// Jidien Kachu Edited in 2025/10/14
FUNCTION_BLOCK FB_RobotAbsMove_V2 EXTENDS FB_ObjectBase_V2 IMPLEMENTS IBasicElement
VAR_INPUT
    Robot         				: REFERENCE TO FB_FanucRobot_Basic_V2;
    LowerConveyor 				: REFERENCE TO FB_Motor;
    // Command   : ST_WareHouseWithRobotMove_Command;
    Info 						: st_AutoSixAxisAbsMoveParameter;
	Input 						: ST_InputTable;
    Stop 						: BOOL;
	Output 						: ST_OutputTable;
	Cylinder 					: REFERENCE TO UNI_CylinderList;
	bCheckUpperCV_ServiceDone	: BOOL;
END_VAR
VAR_OUTPUT
    // Status : ST_WareHouseWithRobotMove_Status;
	AClampMoveDone	: BOOL;
	BClampMoveDone	: BOOL;
END_VAR
VAR
    //_Abort       : BOOL;
    strStatus    : STRING;
    uiResumeStep : UINT;

    Area : E_RobotArea;
    UseA : BOOL;
    UseB : BOOL;

    Get                         : BOOL;
    tonTimeOut                  : TON;
	bTimeOutIN					: BOOL;
	tonDelay					 : TON;
    _UniqueErrorCode            : STRING;
    FirstSensorOfLowerConveyor  : BOOL;
    SecondSensorOfLowerConveyor : BOOL;

	//Added by Jidien Kachu in 2025/10/09
	uiLastBothStep	: UINT;
	uiLastSingleClampStep	: UINT;
	bRobotTimeOutIN	: BOOL;
	tonRobotTimeOut	: TON;
	uiBothStep	: UINT;
	uiSingleClampStep	: UINT;
	bMotorDelayIN	: BOOL;
	tonMotorDelay	: TON;
	bIOTimeoutIN	: BOOL;
	tonIOTimeout	: TON;
	bRetry: BOOL;
	
	//Added by Gamin in 2025//11/24
	_AClampDoingWork	: BOOL;
	_BClampDoingWork	: BOOL;
END_VAR

SUPER^.A10_StateControl();
A00_BasicUnits();
FirstSensorOfLowerConveyor := Input.bLowCV_BoxArrived_Sensor;
SecondSensorOfLowerConveyor := NOT Input.bLowCV_2ndBoxGap_Sensor;// .bLowCV_Block2Detect_Sensor;

(*============================================================
Create Date : 2025/11/22
Last Update	: 2026/04/01
Change Log  : 2025/11/24，send flag A clamp done and B clamp done for C# use to SQL // Edited : Gamin
			  2026/04/01，移植泰興鏡射機版本。
============================================================*)

ACTION A00_BasicUnits:
tonTimeOut(IN:= bTimeOutIN AND NOT THIS^.Stop, PT:=T#60S);
tonDelay(PT:=T#1S);
ErrorID :=2200;
tonMotorDelay(IN:= bMotorDelayIN,PT:=T#1S);
tonIOTimeout(IN:= bIOTimeoutIN,PT:= T#1S);
END_ACTION

METHOD M_CheckClampStatus : BOOL
VAR_INPUT
END_VAR
M_CheckClampStatus := FALSE;

IF NOT UseA AND NOT UseB THEN
	M_CheckClampStatus 	:= FALSE;
	strStatus 			:= 'FB_RobotAbsMove_V2 ,Wrong Command , Both Clammp not used';
	RETURN;
END_IF

IF UseA THEN
	IF Get THEN
		IF NOT Robot._DI1.ClampA_Open THEN
			M_CheckClampStatus  := FALSE;
			strStatus			:= 'FB_RobotAbsMove_V2 ,Robot Use A Clamp Get ,but Clamp not open ';
			RETURN;
		END_IF
	ELSE
		IF Robot._DI1.ClampA_Open THEN
			M_CheckClampStatus	:= FALSE;
			strStatus			:= 'FB_RobotAbsMove_V2 ,Robot Use A Clamp Place ,but Clamp open';
			RETURN;
		END_IF
	END_IF
END_IF
IF UseB THEN
	IF Get THEN
		IF NOT Robot._DI1.ClampB_Open THEN
			M_CheckClampStatus  := FALSE;
			strStatus			:= 'FB_RobotAbsMove_V2 ,Robot Use B Clamp Get ,but Clamp not open ';
			RETURN;
		END_IF
	ELSE
		IF Robot._DI1.ClampB_Open THEN
			M_CheckClampStatus	:= FALSE;
			strStatus			:= 'FB_RobotAbsMove_V2 ,Robot Use B Clamp Place ,but Clamp open';
			RETURN;
		END_IF
	END_IF
END_IF

M_CheckClampStatus := TRUE;
END_METHOD

METHOD M_CheckCommand : BOOL // True : Command is useful
VAR_INPUT
END_VAR
VAR
	
END_VAR
// Check command paremeter is correct


IF Info.A_Get <> Info.B_Get THEN
	strStatus:='Wrong command ,GetA not match to GetB';
	M_CheckCommand:=FALSE;
	RETURN;
ELSE		
	THIS^.Get :=Info.A_Get;
END_IF

IF Info.A_Area<> Info.B_Area THEN
	IF NOT(Info.A_Area=99 OR Info.B_Area=99) THEN
	strStatus:='Wrong command ,Area A not match to Area B';
	M_CheckCommand:=FALSE;
	RETURN;
END_IF
END_IF

IF Info.A_Area = 99 AND Info.B_Area = 99 THEN
	strStatus:='Wrong command ,Both Area are 99';
	M_CheckCommand:=FALSE;
	RETURN;
END_IF

CASE LREAL_TO_INT(Info.A_Area) OF
	1 : //Normal command : RoundBelt
		IF Info.A_Position<1 OR  Info.A_Position>3 THEN
			strStatus:='Wrong command ,Position A Not allow';
			M_CheckCommand:=FALSE;
			RETURN;	
		ELSE
			Area := E_RobotArea.RoundBelt;
			UseA :=TRUE	;	
		END_IF
		
	2:	//Buffer area
		IF Info.A_Position<1 OR  Info.A_Position>40 THEN
			strStatus:='Wrong command ,Position A Not allow';
			M_CheckCommand:=FALSE;
			RETURN;	
		ELSE
			Area := E_RobotArea.BufferArea;
			UseA :=TRUE	;	
		END_IF
	3: //Allocated/Empty conveyor
		IF Info.A_Position<1 OR  Info.A_Position>2 THEN
			strStatus:='Wrong command ,Position A Not allow';
			M_CheckCommand:=FALSE;
			RETURN;	
		ELSE
			Area := E_RobotArea.TransmitCV;
			UseA :=TRUE	;	
		END_IF
	5: //FeedIn/Out conveyor
		IF Info.A_Position<1 OR  Info.A_Position>5 THEN
			strStatus:='Wrong command ,Position A Not allow';
			M_CheckCommand:=FALSE;
			RETURN;	
		ELSIF Info.A_Position=3 AND Get THEN
			strStatus:='Wrong command ,Can Not Get box from FeedOut conveyor ';
			M_CheckCommand:=FALSE;
			RETURN;	
		ELSE
			Area := E_RobotArea.InOutConveyor;
			UseA :=TRUE	;	
		END_IF
	7: // PullOut conveyor
		IF Info.A_Position<1 OR  Info.A_Position>2 THEN
			strStatus:='Wrong command ,Position A Not allow';
			M_CheckCommand:=FALSE;
			RETURN;	
		ELSE
			Area := E_RobotArea.PullOutConveyor;
			UseA :=TRUE	;	
		END_IF
	
	99: //ClampA not use
		UseA :=FALSE;
	
	ELSE //Wrong command
		strStatus:='Wrong command ,Area_A not allow ';
		M_CheckCommand:=FALSE;
		RETURN;

END_CASE

CASE LREAL_TO_INT(Info.B_Area) OF
	1 : //Normal command : RoundBelt
		IF Info.B_Position<1 OR  Info.B_Position>3 THEN
			strStatus:='Wrong command ,Position B Not allow';
			M_CheckCommand:=FALSE;
			RETURN;	
		ELSE
			Area := E_RobotArea.RoundBelt;
			UseB :=TRUE	;	
		END_IF
		
	2:	
		IF Info.B_Position<1 OR  Info.B_Position>40 THEN
			strStatus:='Wrong command ,Position B Not allow';
			M_CheckCommand:=FALSE;
			RETURN;	
		ELSE
			Area := E_RobotArea.BufferArea;
			UseB :=TRUE	;	
		END_IF
	3:
		IF Info.B_Position<1 OR  Info.B_Position>2 THEN
			strStatus:='Wrong command ,Position B Not allow';
			M_CheckCommand:=FALSE;
			RETURN;	
		ELSE
			Area := E_RobotArea.TransmitCV;
			UseB :=TRUE	;	
		END_IF
	5:
		IF Info.B_Position<1 OR  Info.B_Position>5 THEN
			strStatus:='Wrong command ,Position B Not allow';
			M_CheckCommand:=FALSE;
			RETURN;	
		ELSE
			Area := E_RobotArea.InOutConveyor;
			UseB :=TRUE	;	
		END_IF
	7:
		IF Info.B_Position<1 OR  Info.B_Position>2 THEN
			strStatus:='Wrong command ,Position B Not allow';
			M_CheckCommand:=FALSE;
			RETURN;	
		ELSIF Info.B_Position=3 AND Get THEN
			strStatus:='Wrong command ,Can Not Get box from FeedOut conveyor ';
			M_CheckCommand:=FALSE;
			RETURN;	
		ELSE
			Area := E_RobotArea.PullOutConveyor;
			UseB :=TRUE	;	
		END_IF
	
	99: //ClampA not use
		UseB :=FALSE;
	
	ELSE //Wrong command
		strStatus:='Wrong command ,Area_B not allow ';
		M_CheckCommand:=FALSE;
		RETURN;

END_CASE


M_CheckCommand:=TRUE;
END_METHOD

METHOD M_CheckUnitsNotBusy : BOOL
VAR_INPUT
END_VAR
M_CheckUnitsNotBusy := true;
END_METHOD

METHOD M_CheckUnitsReady : BOOL
VAR_INPUT
END_VAR
M_CheckUnitsReady := true;
END_METHOD

METHOD  M_STATE_ABORTED
VAR_INPUT
END_VAR

//Edited by Jidien Kachu in 2025/10/28
IF NOT bRetry THEN
	ERROR :=TRUE;
	Busy    := FALSE;
	Aborted := TRUE;
	Status := strStatus;
	UniqueErrorCode:=_UniqueErrorCode;
	uiAbortingStep := 0;
	_AbortCompleted:=FALSE;//Edited by Jidien Kachu in 2025/10/14
END_IF

IF Reset THEN
	bRetry := TRUE;
	ERROR :=FALSE;
	Aborted := FALSE;
END_IF
IF NOT Execute THEN
	eSTATE:=STATE_RESETTING;
END_IF

IF Execute AND bRetry AND NOT Robot.Error AND NOT Robot.Halt THEN
	uiExecutingStep :=uiResumeStep;

	//Edited by Jidien Kachu in 2025/10/14
	uiBothStep := uiLastBothStep;
	uiSingleClampStep := uiLastSingleClampStep;
	Status := '';


	//////////////////////////////////////
	IF GVL_ADS.MachineState <>E_MachineState.Error THEN
		eSTATE:=STATE_EXECUTING;
	END_IF
END_IF
END_METHOD

METHOD  M_STATE_ABORTING
VAR_INPUT
END_VAR
CASE uiAbortingStep OF
	0 :
			tonDelay.IN 	   := FALSE;
			bTimeOutIN  	   := FALSE;
			tonRobotTimeOut.IN := FALSE;
			_Abort 			   := FALSE;
			bRetry			   := FALSE;
			//Edited by Jidien Kachu in 2025/10/14
			LowerConveyor.M_MotorStop();
			IF 	LowerConveyor.InStopped THEN
				uiAbortingStep:=100;
			END_IF
    100:
			IF Robot._DI1.Error THEN
				uiAbortingStep := 200;
			ELSE
				uiAbortingStep := 9999;
			END_IF
	200:		
			 IF DAS_CoreSys.MachineControl.M_RobotResetCmd() THEN
				 uiAbortingStep := 300;
			 END_IF
	300:
			IF DAS_CoreSys.MachineControl.M_RobotStartCmd() THEN
				 uiAbortingStep := 400;
			 END_IF 
	400:
			IF Robot._DI1.Error THEN
		 		uiAbortingStep := 200;
			ELSE
				uiAbortingStep := 9999;
			END_IF
	
	9999:	
			_AbortCompleted:=TRUE;
END_CASE

IF _AbortCompleted THEN	
	eSTATE :=STATE_ABORTED;
END_IF
END_METHOD

METHOD  M_STATE_DONE
VAR_INPUT
END_VAR
Busy := FALSE;
Done := TRUE;
IF NOT Execute THEN
    eState := STATE_RESETTING;
END_IF
END_METHOD

METHOD  M_STATE_DORMANT
VAR_INPUT
END_VAR
// Clear FB output
Busy            := FALSE;
Done            := FALSE;
Aborted         := FALSE;
Error           := FALSE;
ErrorID         := 0;
Status          := '';
_ResetCompleted := FALSE;
_AbortCompleted := FALSE;
_Error          := FALSE;
_Executed       := FALSE;
tonDelay.IN := FALSE	;
bTimeOutIN:=FALSE;
strStatus :='No Error';
uiExecutingStep :=uiResettingStep :=uiResumeStep :=0;
AClampMoveDone	:= FALSE;
BClampMoveDone	:= FALSE;
_AClampDoingWork	:= FALSE;
_BClampDoingWork	:= FALSE;
bRetry := FALSE;

// Wait Execute command
IF Execute AND NOT stop THEN
    eState := STATE_EXECUTING;
END_IF
END_METHOD

METHOD  M_STATE_ERROR
VAR_INPUT
END_VAR
ERROR   :=TRUE;
Busy	:=FALSE;
Status := strStatus;
UniqueErrorCode:=_UniqueErrorCode;
ErrorID :=2200;

IF NOT Execute THEN	
	eSTATE:=STATE_RESETTING;
END_IF
END_METHOD

METHOD  M_STATE_EXECUTING
VAR_INPUT
END_VAR
VAR_INST
    ActionMode       : E_ReloadRoundBoxAction;
	BoxReady_1st : BOOL;
	BoxReady_2nd : BOOL;
    CarrierReady_1st : BOOL;
    CarrierReady_2nd : BOOL;
    uiBothStep : UINT;
    uiSingleClampStep : UINT;	
	Area : E_RobotArea;
	Address_A : INT;
	Address_B : INT;
END_VAR
VAR
	WareHouse: INT;
END_VAR
// Set Busy active edit by johnson
Busy := TRUE;
(*IF THIS^.Stop THEN // Pending the timeout when Stop signal occur
	tonTimeout.IN :=FALSE;
END_IF*)
// Service Process
CASE uiExecutingStep OF
	0:
        // Clear variable
        ActionMode       := E_ReloadRoundBoxAction.Undefined;
        CarrierReady_1st := FALSE;
        CarrierReady_2nd := FALSE;
//        uiBothStep := 0;
//		uiSingleClampStep :=0;
		uiLastBothStep := 0;//Edited by Jidien Kachu in 2025/10/14
		uiLastSingleClampStep := 0;//Edited by Jidien Kachu in 2025/10/14
		BoxReady_1st := 0;
		BoxReady_2nd := 0;
		bTimeOutIN:=FALSE;
        // Check command
        IF M_CheckCommand() THEN
            uiExecutingStep := 10;
		ELSE
			_Error:=TRUE;
        END_IF
    10:
        // Start process, check units first
        IF M_CheckUnitsReady() THEN
            uiExecutingStep := 20;
        END_IF
    20:
        // CHeck units not busy state
        IF M_CheckUnitsNotBusy() THEN
            uiExecutingStep := 30;
        END_IF
	30:
		IF M_CheckClampStatus() THEN
            uiExecutingStep := 1000;
		ELSE
			_Abort := TRUE;
        END_IF
   
	1000:   
			// Read   coordinate
			 Area := THIS^.Area;
 			 Address_A := LREAL_TO_INT(Info.A_Position);
			 Address_B := LREAL_TO_INT(Info.B_Position);
			 
			IF UseA AND NOT UseB THEN
				//Only clampA
				uiExecutingStep := 10000;
			ELSIF NOT UseA AND UseB THEN
				//Only ClampB 
				uiExecutingStep := 20000;
			ELSIF UseA AND UseB THEN
				//Both Clamps
				uiExecutingStep := 30000;		
			END_IF
       
    10000: // Only ClampA 
        IF NOT Robot._DI1.Done THEN
            //Edited by Jidien Kachu in 2025/10/14
				CASE uiSingleClampStep OF
					0://
						IF Area= E_RobotArea.InOutConveyor AND Address_A=3 THEN
							IF Cylinder.List.fbLowCV_Block1.InRearPosition THEN
								uiSingleClampStep:=100;// Need to control feedout conveyor
							ELSE
								_Error := TRUE;
								strStatus := 'FB_RobotAbsMove_V2 Step 10000: Block 2 cylinder inrearPosition';
							END_IF
						ELSE
							uiSingleClampStep:=1000;	
						END_IF
					100:	
						tonDelay.IN := FALSE	;
						LowerConveyor.M_MoveBackward();
						IF (NOT FirstSensorOfLowerConveyor) AND (NOT SecondSensorOfLowerConveyor) THEN
							bTimeOutIN:=FALSE;;
							uiSingleClampStep:=150;
						END_IF
						bTimeOutIN:=TRUE;
						//Edited by Jidien Kachu in 2025/10/14
						IF tonTimeOut.Q=TRUE OR robot._DI1.Error THEN
							strStatus :='FB_RobotAbsMove_V2 Step 10000: Empty Conveyor timeout';
	//						_Error:=TRUE;
							_Abort := TRUE;
							uiLastSingleClampStep := 0;
							uiResumeStep := 10000;
							uiAbortingStep := 0;
						END_IF
						//////////////////////////////////////////
					150:
						tonDelay.IN := TRUE;
						IF tonDelay.Q THEN
							uiSingleClampStep:=200;
						END_IF	
					200:
						tonDelay.IN := FALSE	;
						LowerConveyor.M_MotorStop();
						uiSingleClampStep:=300;
					
					300:
						IF 	LowerConveyor.InStopped THEN
							bTimeOutIN:=FALSE;
							BoxReady_1st:=TRUE;
							uiSingleClampStep:=9999;
						END_IF
						bTimeOutIN:=TRUE;
						//Edited by Jidien Kachu in 2025/10/14
						IF tonTimeOut.Q=TRUE OR Robot._DI1.Error THEN
							strStatus :='FB_RobotAbsMove_V2 Step 10000: Stop Conveyor timeout';
	//						_Error:=TRUE;
							_Abort := TRUE;
							uiLastSingleClampStep := 200;
							uiResumeStep := 10000;
							uiAbortingStep := 0;
						END_IF	
						//////////////////////////////////////////
					1000:
						// 檢查 A爪去夾爪時，要確保上層輸送帶是完成的。
							IF Area= E_RobotArea.InOutConveyor AND Address_A = 2 THEN
								IF bCheckUpperCV_ServiceDone THEN
									BoxReady_1st:=TRUE;
									_AClampDoingWork := TRUE;
									uiSingleClampStep:=9999;
								END_IF
							ELSE
							BoxReady_1st:=TRUE;
							_AClampDoingWork := TRUE;
							uiSingleClampStep:=9999;
							END_IF
					9999: //Wait	
				END_CASE
//			END_IF
			
			          		 
				  // Robot Abs move
           		 Robot.M_StartRobotAbsMove(GetBox:=Get,
											UseClampA:=UseA,
											UseClampB:=UseB,
											Area:=Area,
											ClampA_Address:=Address_A,
											ClampB_Address:=Address_B,
											BoxReady_1:=BoxReady_1st,
											BoxReady_2:=BoxReady_2nd);		

			// robot doing AClamp done
			IF Get THEN
				IF _AClampDoingWork AND NOT Robot._DI1.ClampA_Open THEN
					AClampMoveDone := TRUE;
				END_IF
			ELSE
				IF _AClampDoingWork AND Robot._DI1.ClampA_Open THEN
					AClampMoveDone := TRUE;
				END_IF
			END_IF	  
		
        ELSE
            uiExecutingStep := 10080;
        END_IF
		IF tonRobotTimeOut.Q THEN
			_Abort 		 := TRUE;
			uiResumeStep := 10000;
			strStatus 	 := 'FB_RobotAbsMove_V2 Step 10000: Robot Move timeout';
		END_IF
		IF Robot._DI1.Error THEN
			_Abort		:= TRUE;
			uiResumeStep:= 10000;
			strStatus	:= CONCAT(STR1 := 'FB_RobotAbsMove_V2 Step 10000:',
								  STR2 := Robot.ErrMsg);
        END_IF
		
    10080:
        Robot.M_ResetRobotAbsMove(UseA,UseB); // Clear command and go to place box
		bTimeOutIN:=TRUE;
        IF NOT Robot._DI1.Done THEN
			bTimeOutIN:=FALSE;
            uiExecutingStep := 40000; 
        END_IF
    	IF tonTimeOut.Q=TRUE THEN
			strStatus :='FB_RobotAbsMove_V2 Step 10080: Reset Robot timeout';
			_Error:=TRUE;
		END_IF
		
    
   20000: // Only ClampB
        IF NOT Robot._DI1.Done THEN
				CASE uiSingleClampStep OF
					0://
						IF Area= E_RobotArea.InOutConveyor AND Address_B=3 THEN
							IF Cylinder.List.fbLowCV_Block1.InRearPosition THEN
								uiSingleClampStep:=100;// Need to control feedout conveyor
							ELSE
								_Error := TRUE;
								strStatus := 'FB_RobotAbsMove_V2 Step 20000: Block 2 cylinder inrearPosition';
							END_IF
						ELSE
							uiSingleClampStep:=1000;	
						END_IF
					100:	
						tonDelay.IN := FALSE;
						LowerConveyor.M_MoveBackward();
						IF (NOT FirstSensorOfLowerConveyor) AND (NOT SecondSensorOfLowerConveyor) THEN
							bTimeOutIN:=FALSE;
							uiSingleClampStep:=150;
						END_IF
						bTimeOutIN:=TRUE;
						//Edited by Jidien Kachu in 2025/10/14
						IF tonTimeOut.Q=TRUE OR Robot._DI1.Error THEN
							strStatus :='FB_RobotAbsMove_V2 Step 20000: Empty Conveyor timeout';
							_Abort := TRUE;
							uiLastSingleClampStep := 0;
							uiResumeStep := 20000;
							uiAbortingStep := 0;
						END_IF	
						///////////////////////////////////////////
					150:
						tonDelay.IN := TRUE;
						IF tonDelay.Q THEN
							uiSingleClampStep:=200;
						END_IF	
		
					200:
						tonDelay.IN := FALSE;
						LowerConveyor.M_MotorStop();
						uiSingleClampStep:=300;
					
					300:
						IF 	LowerConveyor.InStopped THEN
							bTimeOutIN:=FALSE;
							BoxReady_2nd:=TRUE;
							uiSingleClampStep:=9999;
						END_IF
						bTimeOutIN:=TRUE;
						//Edited by Jidien Kachu in 2025/10/14
						IF tonTimeOut.Q=TRUE OR Robot._DI1.Error THEN
							strStatus := 'FB_RobotAbsMove_V2 Step 20000: Stop Conveyor timeout';
	//						_Error:=TRUE;
							_Abort := TRUE;
							uiLastSingleClampStep := 200;
							uiResumeStep := 20000;
							uiAbortingStep := 0;
						END_IF	
						///////////////////////////////////////////
					1000:
							// 檢查 A爪去夾爪時，要確保上層輸送帶是完成的。
							IF Area= E_RobotArea.InOutConveyor AND Address_B = 1 THEN
								IF bCheckUpperCV_ServiceDone THEN
									BoxReady_2nd	 := TRUE;
									_BClampDoingWork := TRUE;
									uiSingleClampStep:=9999;
								END_IF
							ELSE
							BoxReady_2nd	 := TRUE;
							_BClampDoingWork := TRUE;
							uiSingleClampStep:=9999;
							END_IF

					
					9999: //Wait			
				END_CASE
//			END_IF
			
			          		 
				  // Robot Abs move
           		 Robot.M_StartRobotAbsMove( GetBox:=Get,
											UseClampA:=UseA,
											UseClampB:=UseB,
											Area:=Area,
											ClampA_Address:=Address_A,
											ClampB_Address:=Address_B,
											BoxReady_1:=BoxReady_1st,
											BoxReady_2:=BoxReady_2nd);	
											
			// robot doing BClamp done
			IF Get THEN
				IF _BClampDoingWork AND NOT Robot._DI1.ClampB_Open THEN 
					BClampMoveDone := TRUE;
				END_IF
			ELSE
				IF _BClampDoingWork AND  Robot._DI1.ClampB_Open THEN 
					BClampMoveDone := TRUE;
				END_IF
			END_IF
											
        ELSE
            uiExecutingStep := 20080;
        END_IF
		IF tonRobotTimeOut.Q THEN
			_Abort 		 := TRUE;
			uiResumeStep := 20000;
			strStatus 	 := 'FB_RobotAbsMove_V2 Step 20000: Robot Move timeout';
		END_IF
		IF Robot._DI1.Error THEN
			_Abort		:= TRUE;
			uiResumeStep:= 20000;
			strStatus	:= CONCAT(STR1 := 'FB_RobotAbsMove_V2 Step 20000:',
								  STR2 := Robot.ErrMsg);
        END_IF
		
    20080:
       Robot.M_ResetRobotAbsMove(UseA,UseB); // Clear command 
        IF NOT Robot._DI1.Done THEN
            uiExecutingStep := 40000; 
        END_IF
		bTimeOutIN:=TRUE;
		IF tonTimeOut.Q=TRUE THEN
			strStatus :='FB_RobotAbsMove_V2 Step 20080: Reset Robot timeout';
			_Error:=TRUE;
		END_IF	
    30000: // Both Clamps
			CASE uiBothStep OF
           		0://	
					BoxReady_1st := FALSE;
					BoxReady_2nd := FALSE;
					IF Area= E_RobotArea.InOutConveyor AND Address_A=3 THEN
						IF Cylinder.List.fbLowCV_Block1.InRearPosition THEN
								uiBothStep:=100;// Need to control feedout conveyor
							ELSE
								_Error := TRUE;
								strStatus := 'FB_RobotAbsMove_V2 Step 30000: Block 1 cylinder inrearPosition';
							END_IF
					ELSE
						uiBothStep:=1000;	
					END_IF
				100:	
					tonDelay.IN := FALSE;
					LowerConveyor.M_MoveBackward();
					bTimeOutIN:=FALSE;
					IF (NOT FirstSensorOfLowerConveyor) AND (NOT SecondSensorOfLowerConveyor) THEN
						uiBothStep:=150;
					END_IF
					bTimeOutIN:=TRUE;
					//Edited by Jidien Kachu in 2025/10/14
					IF tonTimeOut.Q=TRUE OR Robot._DI1.Error THEN
						strStatus :='FB_RobotAbsMove_V2 Step 30000: Empty Robot timeout';
//						_Error:=TRUE;
						_Abort := TRUE;
						uiLastBothStep := 0;
						uiResumeStep := 30000;
						uiAbortingStep := 0;
					END_IF	
					///////////////////////////////////////////					
				150:
					tonDelay.IN := TRUE;
					IF tonDelay.Q THEN
						uiBothStep:=200;
					END_IF	
				
				200:
					tonDelay.IN := FALSE;
					LowerConveyor.M_MotorStop();
					uiBothStep:=300;
				
				300:
					IF 	LowerConveyor.InStopped THEN
						bTimeOutIN:=FALSE;
						BoxReady_1st:=TRUE;
						uiBothStep:=2000;
					END_IF
					bTimeOutIN:=TRUE;
					//Edited by Jidien Kachu in 2025/10/14
					IF tonTimeOut.Q=TRUE OR Robot._DI1.Error THEN
						strStatus :='FB_RobotAbsMove_V2 Step 30000: Stop Robot timeout';
//						_Error:=TRUE;
						_Abort := TRUE;
						uiLastBothStep := 200;
						uiResumeStep := 30000;
						uiAbortingStep := 0;
					END_IF	
					///////////////////////////////////////////					
				1000:
						// 檢查 A爪去夾爪時，要確保上層輸送帶是完成的。
						IF Area= E_RobotArea.InOutConveyor AND Address_A = 2 THEN
							IF bCheckUpperCV_ServiceDone THEN
						BoxReady_1st	 := TRUE;
						_AClampDoingWork := TRUE;
								uiBothStep		 := 2000;
							END_IF
						ELSE
							BoxReady_1st	 := TRUE;
							_AClampDoingWork := TRUE;
							uiBothStep		 := 2000;
						END_IF
						
				2000:
						IF Robot._DI1.Notification THEN
							uiBothStep:=3000;
						END_IF
						//Edited by Jidien Kachu in 2025/10/14
						IF Robot._DI1.Error THEN
							_Abort := TRUE;
							uiLastBothStep := 0;
							uiResumeStep := 30000;
							uiAbortingStep := 0;
							BoxReady_1st:=FALSE;
						END_IF
						/////////////////////////////////////
				3000:
					
					IF Area= E_RobotArea.InOutConveyor AND Address_B=3 THEN
						uiBothStep:=3100;// Need to control feedout conveyor 
					ELSE
						uiBothStep:=9000;	
					END_IF
				3100:	
					tonDelay.IN := FALSE;
					LowerConveyor.M_MoveBackward();
					IF (NOT FirstSensorOfLowerConveyor) AND (NOT SecondSensorOfLowerConveyor) THEN
						bTimeOutIN:=FALSE;
						uiBothStep:=3200;
					END_IF
					bTimeOutIN:=TRUE;
					//Edited by Jidien Kachu in 2025/10/14
					IF tonTimeOut.Q=TRUE OR Robot._DI1.Error THEN
						strStatus :='FB_RobotAbsMove_V2 Step 30000: Empty Robot timeout';
//						_Error:=TRUE;
						_Abort := TRUE;
						uiLastBothStep := 3000;
						uiResumeStep := 30000;
						uiAbortingStep := 0;
					END_IF	
					///////////////////////////////////////////					
				3200:
					tonDelay.IN := TRUE;
					IF tonDelay.Q THEN
						LowerConveyor.M_MotorStop();
						uiBothStep:=3300;
					END_IF	
					
				
				3300:
					bTimeOutIN:=TRUE;
					tonDelay.IN := FALSE;
					IF 	LowerConveyor.InStopped THEN
						bTimeOutIN:=FALSE;
						BoxReady_2nd:=TRUE;
						uiBothStep:=9999;
					END_IF
					
					//Edited by Jidien Kachu in 2025/10/14
					IF tonTimeOut.Q=TRUE OR Robot._DI1.Error THEN
						strStatus :='FB_RobotAbsMove_V2 Step 30000: Stop Robot timeout';
//						_Error:=TRUE;
						_Abort := TRUE;
						uiLastBothStep := 3200;
						uiResumeStep := 30000;
						uiAbortingStep := 0;
					END_IF	
					///////////////////////////////////////////					
				9000:
						// 檢查 A爪去夾爪時，要確保上層輸送帶是完成的。
						IF Area= E_RobotArea.InOutConveyor AND Address_B = 1 THEN
							IF bCheckUpperCV_ServiceDone THEN
								BoxReady_2nd	 := TRUE;
								_BClampDoingWork := TRUE;
								uiBothStep:=9999;
							END_IF
						ELSE
						BoxReady_2nd	 := TRUE;
						_BClampDoingWork := TRUE;
						uiBothStep:=9999;
						END_IF
				
				9999: //Wait		
				//Edited by Jidien Kachu in 2025/10/14
						IF Robot._DI1.Error THEN
							_Abort := TRUE;
							uiLastBothStep := 3100;
							uiResumeStep := 30000;
							uiAbortingStep := 0;
							BoxReady_2nd:=FALSE;
						END_IF
						/////////////////////////////////////
			// wait reset
			END_CASE
//		END_IF
		
		  

       	  // Robot Abs move
           		 Robot.M_StartRobotAbsMove( GetBox:=Get,
											UseClampA:=UseA,
											UseClampB:=UseB,
											Area:=Area,
											ClampA_Address:=Address_A,
											ClampB_Address:=Address_B,
											BoxReady_1:=BoxReady_1st,
											BoxReady_2:=BoxReady_2nd);	
			IF Get THEN								
				IF _AClampDoingWork AND  NOT Robot._DI1.ClampA_Open THEN
					AClampMoveDone := TRUE;
				END_IF
				IF _BClampDoingWork AND NOT Robot._DI1.ClampB_Open THEN 
					BClampMoveDone := TRUE;
				END_IF
			ELSE
				IF _AClampDoingWork AND Robot._DI1.ClampA_Open THEN
					AClampMoveDone := TRUE;
				END_IF
				IF _BClampDoingWork AND Robot._DI1.ClampB_Open THEN 
					BClampMoveDone := TRUE;
				END_IF
			END_IF
		
		
        IF Robot._DI1.Done THEN
            uiExecutingStep := 30080;
        END_IF
		IF tonRobotTimeOut.Q THEN
			_Abort 		 := TRUE;
			uiResumeStep := 30000;
			strStatus 	 := 'FB_RobotAbsMove_V2 Step 30000: Robot Move timeout';	
		END_IF
		IF Robot._DI1.Error THEN
			_Abort		:= TRUE;
			uiResumeStep:= 30000;
			strStatus	:= CONCAT(STR1 := 'FB_RobotAbsMove_V2 Step 30000:',
								  STR2 := Robot.ErrMsg);
        END_IF
		
    30080: // Check robot command is clear
        
        Robot.M_ResetRobotAbsMove(UseA,UseB);

        IF NOT Robot._DI1.Done THEN
			bTimeOutIN:=FALSE;
			IF Get THEN
				uiExecutingStep := 99000;
			ELSE
				uiExecutingStep := 40000; // go to place step
			END_IF
            
        END_IF    
   		//bTimeOutIN:=TRUE;
		IF tonTimeOut.Q=TRUE THEN
			strStatus := 'FB_RobotAbsMove_V2 Step 30000: Stop Robot timeout';
			_Error:=TRUE;
		END_IF

	40000: // Recheck lowerconveyor Sensor not have box ## Edit by Min 20250416
			
			IF  FirstSensorOfLowerConveyor OR SecondSensorOfLowerConveyor THEN
				bTimeOutIN:=FALSE;
				LowerConveyor.M_MoveBackward();
				uiExecutingStep:=40100;
			ELSE
				uiExecutingStep:=99000;
			END_IF
			bTimeOutIN:=TRUE;
			IF tonTimeOut.Q=TRUE THEN
				strStatus := 'FB_RobotAbsMove_V2 Step 40000: Lowerconveyor Reverse timeout';
				//Edited by Jidien Kachu in 2025/10/14
//				_Error:=TRUE;
				_Abort := TRUE;
				uiResumeStep := 40000;
				uiAbortingStep := 0;
				//////////////////////////////////////
			END_IF	
			
	40100:
			IF NOT (FirstSensorOfLowerConveyor) AND (NOT SecondSensorOfLowerConveyor) THEN
				bTimeOutIN:=FALSE;
				LowerConveyor.M_MotorStop();
				IF LowerConveyor.InStopped THEN
				uiExecutingStep:=99000;
				END_IF
			END_IF
			bTimeOutIN:=TRUE;
			IF tonTimeOut.Q=TRUE THEN
				strStatus :='FB_RobotAbsMove_V2 Step 40100: Lowerconveyor Reverse Stop timeout';
				//Edited by Jidien Kachu in 2025/10/14
//				_Error:=TRUE;
				_Abort := TRUE;
				uiResumeStep := 40100;
				uiAbortingStep := 0;
				//////////////////////////////////////
			END_IF
   
    99000: // process done
        Status    := 'Process completed';
		Cylinder.List.fbLowCV_Block1.M_Retract();
		Cylinder.List.fbLowCV_Press4.M_Retract();
		IF Cylinder.List.fbLowCV_Block1.InRearPosition AND 
			Cylinder.List.fbLowCV_Press4.InRearPosition THEN
			_Executed := TRUE;
			uiBothStep := 0;
			uiSingleClampStep := 0;
		END_IF
END_CASE
IF _Executed THEN
    eState := STATE_DONE;
	uiLastBothStep := 0; //Edited by Jidien Kachu in 2025/10/14
	uiLastSingleClampStep := 0; //Edited by Jidien Kachu in 2025/10/1
ELSIF _Error THEN
	//(iErrorID := ErrorID,UinqueErrorCode=>_UniqueErrorCode);
    eState := STATE_ERROR;
ELSIF NOT Execute THEN
    eState := STATE_RESETTING;
END_IF
IF _Abort OR Abort THEN
	//FUN_UniqueErrorCodeGenerator(iErrorID := ErrorID,UinqueErrorCode=>_UniqueErrorCode);
	eSTATE:=STATE_ABORTING;
END_IF
END_METHOD

METHOD  M_STATE_RESETTING
VAR_INPUT
END_VAR
Error :=FALSE;
Done :=FALSE;
Busy := FALSE;


CASE uiResettingStep OF
	
	0:
		bTimeOutIN:=FALSE;
		tonDelay.IN := FALSE	;
		Robot.M_ResetAllCommand();
		Robot.M_ResetRobotAbsMove(TRUE,TRUE);
		uiResettingStep:=100;
		AClampMoveDone	:= FALSE;
		BClampMoveDone	:= FALSE;
		_AClampDoingWork	:= FALSE;
		_BClampDoingWork	:= FALSE;
		
	100:
		
		LowerConveyor.M_MotorStop();	
		uiResettingStep:=9999;
	9999:
		_ResetCompleted:=TRUE;
END_CASE
IF _ResetCompleted THEN
	eSTATE:=STATE_DORMANT;
END_IF
END_METHOD

END_FUNCTION_BLOCK

(* stored: Version 1.1.0.1, ProductVersion 3.1.4024.13
   POU FB_RobotAbsMove_V2: Id {96b46224-f080-45cd-b7ec-bdd2d780f4c4}, SpecialFunc None
   Folder Method: Id {782c9af9-4f03-469f-9da8-6f4880765cda}
   Folder State: Id {9c458270-fe39-4e17-a2e7-35cffc26ff98}
   Action A00_BasicUnits: Id {50d3543e-42e1-4290-9b06-6917d63c55c6}
   Method M_CheckClampStatus: Id {0189aaaf-bade-4b6a-9182-da0513f60f23}
   Method M_CheckCommand: Id {085c7649-db04-4e86-b7a9-89d9ddef656e}
   Method M_CheckUnitsNotBusy: Id {2b7f4f5a-91f7-47d9-a253-ed4e4f3bd632}
   Method M_CheckUnitsReady: Id {ff3f00d7-8b3d-4a5f-98ec-0f4d2158f48f}
   Method M_STATE_ABORTED: Id {3e2ec5bf-f067-4e19-a33e-84fcdee0fc89}
   Method M_STATE_ABORTING: Id {de2c294e-8a42-414d-96c0-8f06e98c6069}
   Method M_STATE_DONE: Id {0f28394e-e8fe-494a-8d22-1fbe30bbce8d}
   Method M_STATE_DORMANT: Id {249adeba-60cd-40f1-8fb0-853548d8e5a6}
   Method M_STATE_ERROR: Id {35d1104c-9136-41f2-ae5e-534fe447aa33}
   Method M_STATE_EXECUTING: Id {c1985310-0213-4a0c-82e2-a03ba18ac3a3}
   Method M_STATE_RESETTING: Id {886bfdee-0951-452e-9774-96c1d156df6f} *)
